PROGRAM ConfirmableAlarmWithArguments
VAR
	bIsInitialized : BOOL;
	fbAlarm : FB_TcAlarm;
	bRaiseAlarm : BOOL;
	bClearAlarm : BOOL;
	bConfirmAlarm : BOOL;
END_VAR

IF NOT bIsInitialized THEN
	bIsInitialized := TRUE;
	fbAlarm.CreateEx(TC_Events.AlarmsAndEvents.Stop, TRUE, 0);
END_IF

IF bRaiseAlarm THEN
	bRaiseAlarm := FALSE;
	fbAlarm.ipArguments.Clear().AddString('Alice');
	fbAlarm.Raise(0);
END_IF

IF bConfirmAlarm THEN
	bConfirmAlarm := FALSE;
	fbAlarm.Confirm(0);
END_IF

IF bClearAlarm THEN
	bClearAlarm := FALSE;
	fbAlarm.Clear(0, FALSE);
END_IF

END_PROGRAM

(* stored: Version 1.1.0.1, ProductVersion 3.1.4024.12
   POU ConfirmableAlarmWithArguments: Id {dc15ed02-b234-47d5-827f-751c1c4fe3d6}, SpecialFunc None *)
